FUNCTION_BLOCK FB_StateDisabled
VAR_IN_OUT
	stAxis  : ARRAY [GVL.cXP .. GVL.cXM] OF ST_AxisGroup;
	bTopentry : BOOL;
END_VAR
VAR_OUTPUT
	nSMState	: DINT;
END_VAR
VAR_INPUT

END_VAR

IF bTopEntry = TRUE THEN
	bTopEntry := FALSE;
END_IF	
	
stAxis[GVL.cXP].mcPower(Axis := stAxis[GVL.cXP].axisRef, Enable_Positive := FALSE, Enable_Negative := FALSE);
stAxis[GVL.cXM].mcPower(Axis := stAxis[GVL.cXM].axisRef, Enable_Positive := FALSE, Enable_Negative := FALSE);	
stAxis[GVL.cXP].mcHome(Axis := stAxis[GVL.cXP].axisRef, Execute := FALSE);
stAxis[GVL.cXM].mcHome(Axis := stAxis[GVL.cXP].axisRef, Execute := FALSE);
stAxis[GVL.cXP].mcReset(Axis := stAxis[GVL.cXP].axisRef, Execute := FALSE);
stAxis[GVL.cXM].mcReset(Axis := stAxis[GVL.cXM].axisRef, Execute := FALSE);
stAxis[GVL.cXP].bBrake 	:= GVL.cBrakeOn;
stAxis[GVL.cXM].bBrake 	:= GVL.cBrakeOn;
GVL.fbWaitTimer(IN:=FALSE);

nSMState := 10000;

END_FUNCTION_BLOCK

(* stored: Version 1.1.0.1, ProductVersion 3.1.4020.12
   POU FB_StateDisabled: Id {d1cd4ba5-bb4f-4099-a180-cb41c9ee3f71}, SpecialFunc None *)
